FUNCTION_BLOCK CallButton (* Composite Function Block Type *)
  (* Standard: 61499-2 *)
  (* Version 0.0, 6/3/2016, Andrei, nxtControl GmbH, template *)
  PACKAGE Main;
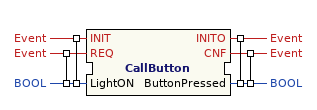
  EVENT_INPUT
    INIT WITH LightON; (* Initialization Request *)
    REQ WITH LightON; (* Normal Execution Request *)
  END_EVENT
  EVENT_OUTPUT
    INITO WITH ButtonPressed; (* Initialization Confirm *)
    CNF WITH ButtonPressed; (* Execution Confirmation *)
  END_EVENT
  VAR_INPUT
    LightON : BOOL; (* Input event qualifier *)
  END_VAR
  VAR_OUTPUT
    ButtonPressed : BOOL; (* Output event qualifier *)
  END_VAR
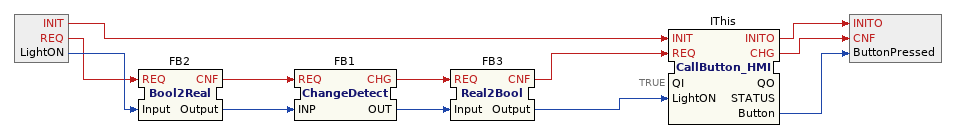
  FBS
    IThis : CallButton_HMI(QI := TRUE);
    FB1 : ChangeDetect;
    FB2 : Bool2Real;
    FB3 : Real2Bool;
  END_FBS
  EVENT_CONNECTIONS
    REQ TO FB2.REQ;
    FB1.CHG TO FB3.REQ;
    FB2.CNF TO FB1.REQ;
    INIT TO IThis.INIT;
    FB3.CNF TO IThis.REQ;
    IThis.INITO TO INITO;
    IThis.CHG TO CNF;
  END_CONNECTIONS
  DATA_CONNECTIONS
    LightON TO FB2.Input;
    FB1.OUT TO FB3.Input;
    FB2.Output TO FB1.INP;
    FB3.Output TO IThis.LightON;
    IThis.Button TO ButtonPressed;
  END_CONNECTIONS
END_FUNCTION_BLOCK
